(*********************************** G.D S.p.A. - Technical Department ***********************************
============= PROGRAM INFO ============
FOLDER:             TBD
MACHINES INVOLVED:  TBD 

============= DESCRIPTION =============
csp machine declaration

============= REVISIONS ===============
Date		Version	 	Author      	Description             
----------	-------		------------  	--------------------------------------------
2019/04/05 	0000.00	 	M.Grasso		Creation of the PRG

**********************************************************************************************************)
(*$R process_ref := prc; $*)
PROGRAM csp_case_fc_ls_lower
VAR
	
	prc:											process;
	prc_path:										STRING;
	
END_VAR

_read_var_input();

_object_manager();

IF NOT objects_running()
THEN
	RETURN;	
END_IF

_read_process_image();

_mode_manager();

_set_runtime_properties();

(********************************* BODY *********************************)
(************************************************************************)

_handle_messages();

_write_output();

ACTION _handle_messages:
;
END_ACTION

ACTION _handle_process_test:
;
END_ACTION

ACTION _mode_manager:
IF process_mode_req_is_pending(prc)
THEN
    process_apply_mode_req_first_step(prc);
    CASE process_get_mode(prc) OF
        MODE_TO_ABSENT:
			;
        MODE_TO_INACTIVE:
			;
        MODE_TO_TEST:
			;
        MODE_TO_OPERATIONAL:
			;
    END_CASE
    process_apply_mode_req_second_step(prc);
END_IF
END_ACTION

ACTION _object_manager:
IF objects_initialization()
THEN
	sub_process_init(
		object_name					:= 'csp_case_fc_ls_lower.prc', 
		process						:= csp_case_flapControl_ls.prc, 
		CONVERSION_this				:= prc);
		
	prc_path 						:= process_get_path(prc);
END_IF

IF objects_running()
THEN
	process_cycle(prc);
END_IF
END_ACTION

ACTION _read_process_image:
;
END_ACTION

ACTION _read_var_input:
;
END_ACTION

ACTION _set_runtime_properties:
;
END_ACTION

ACTION _write_output:
;
END_ACTION

END_PROGRAM

(* stored: Version 1.1.0.1, ProductVersion 3.1.4022.12
   POU csp_case_fc_ls_lower: Id {3b7eba9a-6156-438f-9601-47bfe9615ff0}, SpecialFunc None
   Action _handle_messages: Id {c337a9ab-14ae-455f-8a11-259e8aa6c101}
   Action _handle_process_test: Id {fd7aecef-405f-4302-8337-11d2238f03d8}
   Action _mode_manager: Id {9fb5e5d6-2904-4787-bd31-3ba871d70aea}
   Action _object_manager: Id {122dbdc1-908b-4755-8c12-beae786228b9}
   Action _read_process_image: Id {07ff6887-ebf3-45b8-930f-aa0e7975a8e3}
   Action _read_var_input: Id {eecc6686-fa02-40cb-9798-6fbb3a530b69}
   Action _set_runtime_properties: Id {625033f1-960e-4334-bf77-0ec4b4dbd4c6}
   Action _write_output: Id {d2357e2d-7924-4576-8a9d-87cfdd70443b} *)
